// TIA Portal V18 export
TYPE "UDT_AIadv"
// stored: IsFailsafeCompliant false
   STRUCT
      rValue : Real;   // Real value
      rMin : Real;   // Scale Min
      rMax : Real;   // Scale Max
      rCalibration : Real;
      iFuncSystemID : Byte := 0;
      iFuncVar : Byte := 0;
      rFilterSet : Real;   // Filter value
   END_STRUCT;
END_TYPE
